# B&R Automation Studio project poarlab1
Automation Studio 4.5.2.102

## Configuration Real

CPU 4PP065.0571-P74, AutomationRuntime D4.52, Build 4.1.2, Vc V4.52.0

### Task classes (Cpu.sw)
```
Cyclic#1:
  Program1 <- Program1.prg
Binaries: udbdef, TCData, ashwd, User, asfw, sysconf, arconfig, ashwac, iomap, Role
Libraries: Motor
```

### Hardware
```
4PP065_0571_P74 : 4PP065.0571-P74 v1.1.2.0
  Connector IF5:
    ActivateDevice = 1
  ConfigurationID = laba1_Real
  Simulation = 1
```

## Logical view

Binary libraries used (declarations not repeated): operator, runtime, astime, AsIecCon

### Package Logical/Libraries - Global libraries

### Library Logical/Libraries/Motor (ANSIC)

#### Motor.fun - Exported functions and function blocks
```iecst
{REDUND_ERROR} FUNCTION_BLOCK FB_integrator (*TODO: Add your comment here*) (*$GROUP=User,$CAT=User,$GROUPICON=User.png,$CATICON=User.png*)
	VAR_INPUT
		in : REAL;
	END_VAR
	VAR_OUTPUT
		out : {REDUND_UNREPLICABLE} REAL;
	END_VAR
	VAR
		dt : REAL;
	END_VAR
END_FUNCTION_BLOCK

{REDUND_ERROR} FUNCTION_BLOCK FB_motor (*TODO: Add your comment here*) (*$GROUP=User,$CAT=User,$GROUPICON=User.png,$CATICON=User.png*)
	VAR_INPUT
		u : REAL;
	END_VAR
	VAR_OUTPUT
		w : {REDUND_UNREPLICABLE} REAL;
		phi : {REDUND_UNREPLICABLE} REAL;
	END_VAR
	VAR
		integrator : FB_integrator;
		Tm : REAL;
		ke : REAL;
		dt : REAL;
	END_VAR
END_FUNCTION_BLOCK

{REDUND_ERROR} FUNCTION_BLOCK FB_regulator (*TODO: Add your comment here*) (*$GROUP=User,$CAT=User,$GROUPICON=User.png,$CATICON=User.png*)
	VAR_INPUT
		e : REAL;
	END_VAR
	VAR_OUTPUT
		u : {REDUND_UNREPLICABLE} REAL;
	END_VAR
	VAR
		k_p : REAL;
		k_i : REAL;
		integrator : FB_integrator;
		iyOld : REAL;
		max_abs_value : REAL;
		dt : REAL;
		e_p : REAL;
	END_VAR
END_FUNCTION_BLOCK
```

#### FB_integrator.c
```c
#include <bur/plctypes.h>
#ifdef __cplusplus
	extern "C"
	{
#endif
	#include "Motor.h"
#ifdef __cplusplus
	};
#endif
/* TODO: Add your comment here */
void FB_integrator(struct FB_integrator* inst)
{
	inst->out = inst->out + inst->in;
	/*TODO: Add your code here*/
}
```

#### FB_motor.c
```c
#include <bur/plctypes.h>
#ifdef __cplusplus
	extern "C"
	{
#endif
	#include "Motor.h"
#ifdef __cplusplus
	};
#endif
/* TODO: Add your comment here */
void FB_motor(struct FB_motor* inst)
{
	inst->integrator.in = (inst->u/inst->ke - inst->w) * inst->dt/inst->Tm;
	FB_integrator(&inst->integrator);

	inst->w = inst->integrator.out;

	inst->integrator.in = inst->w*inst->dt;
	FB_integrator(&inst->integrator);
	inst->phi = inst->integrator.out;

	/*TODO: Add your code here*/
}
```

#### FB_regulator.c
```c
#include <math.h>
#include <bur/plctypes.h>
#ifdef __cplusplus
	extern "C"
	{
#endif
	#include "Motor.h"
#ifdef __cplusplus
	};
#endif
/* TODO: Add your comment here */
void FB_regulator(struct FB_regulator* inst)
{
    /*TODO: Add your code here*/
    inst->integrator.in = inst->e*inst->k_i*inst->dt+inst->iyOld;
    FB_integrator(&(inst->integrator));
    inst->e_p = inst->e * inst->k_p;
    if (inst->e_p>inst->max_abs_value || inst->e_p < -inst->max_abs_value) {
        if (inst->e_p>0) inst->e_p = inst->max_abs_value;
        else inst->e_p = -inst->max_abs_value;
    }
    inst->e_p += inst->integrator.out;
    if (inst->e_p<inst->max_abs_value || inst->e_p > -inst->max_abs_value) inst->u = inst->e_p;
    else
    {
        if (inst->e_p>0) inst->u = inst->max_abs_value;
        else inst->u = -inst->max_abs_value;
    }
    inst->iyOld = inst->u - inst->e_p;
}
```

### Program Logical/Program1 (ANSIC)

#### Variables.var
```iecst
VAR
	fb_motor : FB_motor;
	speed : REAL;
	fb_regulator : FB_regulator;
	enable : BOOL;
	fb_motor2 : FB_motor;
	count : REAL;
END_VAR
```

#### Main.c
```c
#include <bur/plctypes.h>

#ifdef _DEFAULT_INCLUDES
	#include <AsDefault.h>
#endif

void _INIT ProgramInit(void)
{
    enable = 1;
    count = 0;
    speed = 0;
    fb_motor.dt = 0.01;
    fb_motor.ke = 0.24;
    fb_motor.Tm = 0.1;
    fb_motor2.dt = 0.01;
    fb_motor2.ke = 0.24;
    fb_motor2.Tm = 0.1;
    fb_regulator.dt = 0.01;
    fb_regulator.k_p = 5;
    fb_regulator.k_i = 3;
    fb_regulator.max_abs_value = 24;

}

void _CYCLIC ProgramCyclic(void)
{
    if (enable == 1){
        count +=10;
        if (count >=400 && count <=2000) speed = 40;
        else{
            speed = 5;
        }
        if (count>=2000){
            count=0;
        }
    }
    else{
        speed = 0;
    }
    fb_regulator.e = speed - fb_motor.w;
    fb_motor2.u = speed * fb_motor2.ke;
    fb_motor.u = fb_regulator.u*fb_motor.ke;
    FB_regulator(&fb_regulator);
    FB_motor(&fb_motor);
    FB_motor(&fb_motor2);

}

void _EXIT ProgramExit(void)
{

}
```

Listed in the project but not available here: Logical/Global.typ, Logical/Global.var, Logical/Libraries/Motor/Types.typ, Logical/Libraries/Motor/Constants.var
